(* IEC 61131-3 sources: ebr_tool/project_scaffold_full/src/helpers, 4 files *)

(* ---- le_helpers.st ---- *)
(******************************************************************)
(*  Little-Endian helpers for spinIF frames                        *)
(******************************************************************)
FUNCTION WriteUInt16LE : UDINT
VAR_INPUT pDst : POINTER TO BYTE;  val : UINT; END_VAR
pDst^ := BYTE(val AND 16#00FF); pDst := pDst + 1;
pDst^ := BYTE(SHR(val,8) AND 16#00FF);
WriteUInt16LE := 2;

FUNCTION WriteInt16LE : UDINT
VAR_INPUT pDst : POINTER TO BYTE;  val : INT; END_VAR
WriteUInt16LE(pDst:=pDst, val:=TO_UINT(val));
WriteInt16LE := 2;

FUNCTION WriteUInt32LE : UDINT
VAR_INPUT pDst : POINTER TO BYTE;  val : UDINT; END_VAR
pDst^ := BYTE(val AND 16#FF);      pDst := pDst + 1;
pDst^ := BYTE(SHR(val,8) AND 16#FF); pDst := pDst + 1;
pDst^ := BYTE(SHR(val,16) AND 16#FF); pDst := pDst + 1;
pDst^ := BYTE(SHR(val,24) AND 16#FF);
WriteUInt32LE := 4;

FUNCTION WriteInt32LE : UDINT
VAR_INPUT pDst : POINTER TO BYTE;  val : DINT; END_VAR
WriteUInt32LE(pDst:=pDst, val:=TO_UDINT(val));
WriteInt32LE := 4;

FUNCTION ReadUInt16LE : UINT
VAR_INPUT pSrc : POINTER TO BYTE; END_VAR
VAR b0,b1: UINT; p: POINTER TO BYTE; END_VAR
p := pSrc; b0 := p^; p := p + 1; b1 := p^; ReadUInt16LE := UINT(b0 OR SHL(b1,8));

FUNCTION ReadInt16LE : INT
VAR_INPUT pSrc : POINTER TO BYTE; END_VAR
ReadInt16LE := TO_INT(ReadUInt16LE(pSrc));

FUNCTION ReadUInt32LE : UDINT
VAR_INPUT pSrc : POINTER TO BYTE; END_VAR
VAR b0,b1,b2,b3: UDINT; p: POINTER TO BYTE; END_VAR
p := pSrc; b0 := p^; p := p + 1; b1 := p^; p := p + 1; b2 := p^; p := p + 1; b3 := p^;
ReadUInt32LE := b0 OR SHL(b1,8) OR SHL(b2,16) OR SHL(b3,24);

FUNCTION ReadInt32LE : DINT
VAR_INPUT pSrc : POINTER TO BYTE; END_VAR
ReadInt32LE := TO_DINT(ReadUInt32LE(pSrc));

(* ---- logger.st ---- *)
(******************************************************************)
(*  Lightweight logger using pers.WarningLog[] ringbuffer         *)
(******************************************************************)
FUNCTION DTG_LogLine : BOOL
VAR_INPUT sLine : STRING; END_VAR
VAR idx : INT; END_VAR
idx := pers.WloggingCounter MOD 300;
pers.WarningLog[idx] := sLine;
pers.WloggingCounter := pers.WloggingCounter + 1;
DTG_LogLine := TRUE;

FUNCTION DTG_NibHex : STRING(1)
VAR_INPUT nib : BYTE; END_VAR
CASE TO_INT(nib) OF
 0: DTG_NibHex:='0'; 1:'1'; 2:'2'; 3:'3'; 4:'4'; 5:'5'; 6:'6'; 7:'7';
 8: '8'; 9:'9'; 10:'A'; 11:'B'; 12:'C'; 13:'D'; 14:'E'; 15:'F';
ELSE DTG_NibHex:='?'; END_CASE

FUNCTION DTG_LogHex : BOOL
VAR_INPUT pBuf: POINTER TO BYTE; udiLen: UDINT; sTitle: STRING; END_VAR
VAR i, maxN: UDINT; b,hi,lo: BYTE; p: POINTER TO BYTE; sLine: STRING(255); END_VAR
sLine := CONCAT(sTitle, ': '); p := pBuf; maxN := 32; IF udiLen < maxN THEN maxN := udiLen; END_IF;
FOR i:=0 TO maxN-1 DO
 b := p^; hi := SHR(b,4) AND 16#0F; lo := b AND 16#0F;
 sLine := CONCAT(sLine, DTG_NibHex(hi)); sLine := CONCAT(sLine, DTG_NibHex(lo));
 IF i < (maxN-1) THEN sLine := CONCAT(sLine,' '); END_IF; p := p + 1;
END_FOR;
DTG_LogLine(sLine); DTG_LogHex := TRUE;

(* ---- interlock_engine.st ---- *)
(******************************************************************)
(*  FB_InterlockEngine – centrale regels                           *)
(******************************************************************)
FUNCTION_BLOCK FB_InterlockEngine
VAR_INPUT
    LID_ClosedLocked : BOOL;
    VAC_Ok           : BOOL;
    EtherCAT_Up      : BOOL;
    Spn_Mode         : BYTE;   // STATcon.spindle.mode
    Spn_dlyEC        : BYTE;   // STATcon.spindle.dlyEC
    StopCond         : DWORD;  // STATcon.err_flg of actuele StopConditions
    Cobot_Ready      : BOOL;
END_VAR
VAR_OUTPUT
    AllowMotion  : BOOL;
    BlockReason  : UINT;   // code voor HMI
END_VAR
VAR
    busy : BOOL;
END_VAR

// Eenvoudige regelset (MVP) – uitbreiden naar behoefte
AllowMotion := TRUE; BlockReason := 0;
IF NOT EtherCAT_Up THEN AllowMotion:=FALSE; BlockReason:=100; END_IF;
IF NOT LID_ClosedLocked THEN AllowMotion:=FALSE; BlockReason:=101; END_IF;
IF NOT VAC_Ok THEN AllowMotion:=FALSE; BlockReason:=102; END_IF;
IF (Spn_Mode = 16#0A) THEN AllowMotion:=FALSE; BlockReason:=103; END_IF; // PSTOP
IF (Spn_dlyEC = 16#16) THEN AllowMotion:=FALSE; BlockReason:=104; END_IF; // BUSY
IF NOT Cobot_Ready THEN AllowMotion:=FALSE; BlockReason:=105; END_IF;
// voorbeeld StopCondition maskers (UVOLT bit2, OVOLT bit3, OVRLD bit5, LID_OPEN bit13)
IF (StopCond AND 16#0000000C) <> 0 THEN AllowMotion:=FALSE; BlockReason:=201; END_IF; // UV/OV
IF (StopCond AND 16#00000020) <> 0 THEN AllowMotion:=FALSE; BlockReason:=202; END_IF; // OVRLD
IF (StopCond AND 16#00002000) <> 0 THEN AllowMotion:=FALSE; BlockReason:=203; END_IF; // LID_OPEN

(* ---- recipe_executor.st ---- *)
(******************************************************************)
(*  FB_RecipeExecutor – eenvoudige sequentie‑executor             *)
(******************************************************************)
FUNCTION_BLOCK FB_RecipeExecutor
VAR_INPUT
    Start     : BOOL;
    Stop      : BOOL;
    Rcp       : RECIPE;   // zie docs/recipe_spec.md
    Allow     : BOOL;     // van interlock engine
END_VAR
VAR_OUTPUT
    Busy      : BOOL;
    Error     : BOOL;
    StepIdx   : UINT;
    Msg       : STRING(120);
END_VAR
VAR
    st : (IDLE, RUN, HOLD, DONE, ABORT);
    t  : TON;
END_VAR

CASE st OF
IDLE:
    IF Start AND Allow AND (Rcp.Count > 0) THEN
        StepIdx := 1; Busy := TRUE; Error := FALSE; Msg := '';
        st := RUN;
    END_IF;
RUN:
    // TODO: dispatch naar devices aan de hand van Rcp.Steps[StepIdx]
    // Placeholder: wacht HoldMs en ga door
    t(IN:=TRUE, PT:=T#100MS);
    IF t.Q THEN
        t(IN:=FALSE); StepIdx := StepIdx + 1;
        IF StepIdx > Rcp.Count THEN st := DONE; END_IF;
    END_IF;
DONE:
    Busy:=FALSE; Msg:='Recipe klaar';
    IF Stop THEN st := IDLE; END_IF;
ABORT:
    Busy:=FALSE; Error:=TRUE; Msg:='Afgebroken';
    IF Stop THEN st := IDLE; END_IF;
END_CASE
